FUNCTION ToTrigger : BOOL
VAR_INPUT
	ipChObject : I_CH_OBJECT;
	ipXtsTrigger : REFERENCE TO I_XTS_Trigger;
END_VAR

VAR
	ipTmp : I_XTS_Trigger;
END_VAR

(* 
   1. Test if the interface exists
   2. Test if the object implements a "Object" interface 
   3. Write reference to interface in parameter
   4. Returne TRUE if succesfull
*)
IF ipChObject <> 0 AND_THEN __QUERYINTERFACE(ipChObject,ipTmp) THEN
	ipXtsTrigger := ipTmp;
	ToTrigger := TRUE;
END_IF

END_FUNCTION

(* stored: Version 1.1.0.1, ProductVersion 3.1.4024.12
   POU ToTrigger: Id {24c06874-f91b-4a65-84e0-1578471928c8}, SpecialFunc None *)
